PROGRAM Recipe13
VAR_INPUT
	ExecutingRecipe1: BOOL;
END_VAR
VAR_OUTPUT
	SuccesfullyEnded: BOOL := FALSE;
END_VAR
VAR
	State: INT := 0;
	WoodInitialLiftingPosition: INT := 50;
	InitialExtensionPosition: INT := 388;
	MaxGripPosition: INT := 160;
	RotationDropOffPosition: INT := 300;
	PlasticsInitialLiftingPosition: INT := 250;
	PlasticsDropOffExtensionPosition: INT := 300;
	MetalInitialLiftingPosition: INT := 400;
	MetalDropOffExtensionPosition: INT := 500;
END_VAR

// Recipe is sequence of moves to execute the task.

IF ExecutingRecipe1 THEN	// we start executing recipe1 (again)
	SuccesfullyEnded := FALSE;
END_IF

IF NOT IO.Switch AND NOT SuccesfullyEnded THEN
	IO.LEDGreen := 1;
	// WOOD:
	IF State = 0 THEN
		IF Automatic.LiftingPositionAuto < WoodInitialLiftingPosition THEN
			IO.MotorLiftingDirection := 0;
			IF NOT Automatic.SafetyLON THEN
				Automatic.MotorL.CurrentlyMoving := TRUE;
				IO.MotorLifting := 1;
			END_IF
		ELSE
			State := 1;
			IO.MotorLifting := 0;
			Automatic.MotorL.CurrentlyMoving := FALSE;
		END_IF
	ELSIF State = 1 THEN
		IF Automatic.ExtensionPositionAuto < InitialExtensionPosition THEN
			IO.MotorExtensionDirection := 0;
			IF NOT Automatic.SafetyEON THEN
				Automatic.MotorE.CurrentlyMoving := TRUE;
				IO.MotorExtension := 1;
			END_IF
		ELSE
			State := 2;
			IO.MotorExtension := 0;
			Automatic.MotorE.CurrentlyMoving := FALSE;
		END_IF
	ELSIF State = 2 THEN
		IF Automatic.GripPositionAuto < MaxGripPosition THEN
			IO.MotorGripDirection := 0;
			IF NOT Automatic.SafetyGON THEN
				Automatic.MotorG.CurrentlyMoving := TRUE;
				IO.MotorGrip := 1;
			END_IF
		ELSE
			State := 3;
			IO.MotorGrip := 0;
			Automatic.MotorG.CurrentlyMoving := FALSE;
		END_IF
	ELSIF State = 3 THEN
		IF NOT IO.EndLiftingSensor THEN
			IO.MotorLiftingDirection := 1;
			IF NOT Automatic.SafetyLON THEN
				Automatic.MotorG.CurrentlyMoving := TRUE;
				IO.MotorLifting := 1;
			END_IF
		ELSE
			State := 4;
			IO.MotorLifting := 0;
			Automatic.MotorL.CurrentlyMoving := FALSE;
		END_IF
	ELSIF State = 4 THEN
		IF Automatic.RotationPositionAuto < RotationDropOffPosition THEN
			IO.MotorRotationDirection := 0;
			IF NOT Automatic.SafetyRON THEN
				Automatic.MotorR.CurrentlyMoving := TRUE;
				IO.MotorRotation := 1;
			END_IF
		ELSE
			State := 5;
			IO.MotorRotation := 0;
			Automatic.MotorR.CurrentlyMoving := FALSE;
		END_IF
	ELSIF State = 5 THEN
		IF NOT IO.EndExtensionSensor THEN	// it drops wood in the nearest bin
			IO.MotorExtensionDirection := 1;
			IF NOT Automatic.SafetyEON THEN
				Automatic.MotorE.CurrentlyMoving := TRUE;
				IO.MotorExtension := 1;
			END_IF
		ELSE
			State := 6;
			IO.MotorExtension := 0;
			Automatic.MotorE.CurrentlyMoving := FALSE;
		END_IF
	ELSIF State = 6 THEN
		IF NOT IO.EndGripSensor THEN
			IO.MotorGripDirection := 1;
			IF NOT Automatic.SafetyGON THEN
				Automatic.MotorG.CurrentlyMoving := TRUE;
				IO.MotorGrip := 1;
			END_IF
		ELSE
			State := 7;
			IO.MotorGrip := 0;
			Automatic.MotorG.CurrentlyMoving := FALSE;
		END_IF
	ELSIF State = 7 THEN
		IF NOT IO.EndRotationSensor THEN
			IO.MotorRotationDirection := 1;
			IF NOT Automatic.SafetyRON THEN
				Automatic.MotorR.CurrentlyMoving := TRUE;
				IO.MotorRotation := 1;
			END_IF
		ELSE
			State := 8;
			IO.MotorRotation := 0;
			Automatic.MotorR.CurrentlyMoving := FALSE;
		END_IF
	END_IF
	
	// PLASTICS:
	IF State = 8 THEN
		IF Automatic.LiftingPositionAuto < PlasticsInitialLiftingPosition THEN
			IO.MotorLiftingDirection := 0;
			IF NOT Automatic.SafetyLON THEN
				Automatic.MotorL.CurrentlyMoving := TRUE;
				IO.MotorLifting := 1;
			END_IF
		ELSE
			State := 9;
			IO.MotorLifting := 0;
			Automatic.MotorL.CurrentlyMoving := FALSE;
		END_IF
	ELSIF State = 9 THEN
		IF Automatic.ExtensionPositionAuto < InitialExtensionPosition THEN
			IO.MotorExtensionDirection := 0;
			IF NOT Automatic.SafetyEON THEN
				Automatic.MotorE.CurrentlyMoving := TRUE;
				IO.MotorExtension := 1;
			END_IF
		ELSE
			State := 10;
			IO.MotorExtension := 0;
			Automatic.MotorE.CurrentlyMoving := FALSE;
		END_IF
	ELSIF State = 10 THEN
		IF Automatic.GripPositionAuto < MaxGripPosition THEN
			IO.MotorGripDirection := 0;
			IF NOT Automatic.SafetyGON THEN
				Automatic.MotorG.CurrentlyMoving := TRUE;
				IO.MotorGrip := 1;
			END_IF
		ELSE
			State := 11;
			IO.MotorGrip := 0;
			Automatic.MotorG.CurrentlyMoving := FALSE;
		END_IF
	ELSIF State = 11 THEN
		IF NOT IO.EndLiftingSensor THEN
			IO.MotorLiftingDirection := 1;
			IF NOT Automatic.SafetyLON THEN
				Automatic.MotorL.CurrentlyMoving := TRUE;
				IO.MotorLifting := 1;
			END_IF
		ELSE
			State := 12;
			IO.MotorLifting := 0;
			Automatic.MotorL.CurrentlyMoving := FALSE;
		END_IF
	ELSIF State = 12 THEN
		IF Automatic.RotationPositionAuto < RotationDropOffPosition THEN
			IO.MotorRotationDirection := 0;
			IF NOT Automatic.SafetyRON THEN
				Automatic.MotorR.CurrentlyMoving := TRUE;
				IO.MotorRotation := 1;
			END_IF
		ELSE
			State := 13;
			IO.MotorRotation := 0;
			Automatic.MotorR.CurrentlyMoving := FALSE;
		END_IF
	ELSIF State = 13 THEN
		IF Automatic.ExtensionPositionAuto > PlasticsDropOffExtensionPosition THEN	// it drops plastics into second nearest bin
			IO.MotorExtensionDirection := 1;
			IF NOT Automatic.SafetyEON THEN
				Automatic.MotorE.CurrentlyMoving := TRUE;
				IO.MotorExtension := 1;
			END_IF
		ELSE
			State := 14;
			IO.MotorExtension := 0;
			Automatic.MotorE.CurrentlyMoving := FALSE;
		END_IF
	ELSIF State = 14 THEN
		IF NOT IO.EndGripSensor THEN
			IO.MotorGripDirection := 1;
			IF NOT Automatic.SafetyGON THEN
				Automatic.MotorG.CurrentlyMoving := TRUE;
				IO.MotorGrip := 1;
			END_IF
		ELSE
			State := 15;
			IO.MotorGrip := 0;
			Automatic.MotorG.CurrentlyMoving := FALSE;
		END_IF
	ELSIF State = 15 THEN
		IF NOT IO.EndRotationSensor THEN
			IO.MotorRotationDirection := 1;
			IF NOT Automatic.SafetyRON THEN
				Automatic.MotorR.CurrentlyMoving := TRUE;
				IO.MotorRotation := 1;
			END_IF
		ELSE
			State := 16;
			IO.MotorRotation := 0;
			Automatic.MotorR.CurrentlyMoving := FALSE;
		END_IF
	END_IF
	
	// METAL:
	IF State = 16 THEN
		IF Automatic.LiftingPositionAuto < MetalInitialLiftingPosition THEN
			IO.MotorLiftingDirection := 0;
			IF NOT Automatic.SafetyLON THEN
				Automatic.MotorL.CurrentlyMoving := TRUE;
				IO.MotorLifting := 1;
			END_IF
		ELSE
			State := 17;
			IO.MotorLifting := 0;
			Automatic.MotorL.CurrentlyMoving := FALSE;
		END_IF
	ELSIF State = 17 THEN
		IF Automatic.ExtensionPositionAuto < InitialExtensionPosition THEN
			IO.MotorExtensionDirection := 0;
			IF NOT Automatic.SafetyEON THEN
				Automatic.MotorE.CurrentlyMoving := TRUE;
				IO.MotorExtension := 1;
			END_IF
		ELSE
			State := 18;
			IO.MotorExtension := 0;
			Automatic.MotorE.CurrentlyMoving := FALSE;
		END_IF
	ELSIF State = 18 THEN
		IF Automatic.GripPositionAuto < MaxGripPosition THEN
			IO.MotorGripDirection := 0;
			IF NOT Automatic.SafetyGON THEN
				Automatic.MotorG.CurrentlyMoving := TRUE;
				IO.MotorGrip := 1;
			END_IF
		ELSE
			State := 19;
			IO.MotorGrip := 0;
			Automatic.MotorG.CurrentlyMoving := FALSE;
		END_IF
	ELSIF State = 19 THEN
		IF NOT IO.EndLiftingSensor THEN
			IO.MotorLiftingDirection := 1;
			IF NOT Automatic.SafetyLON THEN
				Automatic.MotorL.CurrentlyMoving := TRUE;
				IO.MotorLifting := 1;
			END_IF
		ELSE
			State := 20;
			IO.MotorLifting := 0;
			Automatic.MotorL.CurrentlyMoving := FALSE;
		END_IF
	ELSIF State = 20 THEN
		IF Automatic.RotationPositionAuto < RotationDropOffPosition THEN
			IO.MotorRotationDirection := 0;
			IF NOT Automatic.SafetyRON THEN
				Automatic.MotorR.CurrentlyMoving := TRUE;
				IO.MotorRotation := 1;
			END_IF
		ELSE
			State := 21;
			IO.MotorRotation := 0;
			Automatic.MotorR.CurrentlyMoving := FALSE;
		END_IF
	ELSIF State = 21 THEN
		IF Automatic.ExtensionPositionAuto > MetalDropOffExtensionPosition THEN	// it drops metal into farthest bin
			IO.MotorExtensionDirection := 1;
			IF NOT Automatic.SafetyEON THEN
				Automatic.MotorE.CurrentlyMoving := TRUE;
				IO.MotorExtension := 1;
			END_IF
		ELSE
			State := 22;
			IO.MotorExtension := 0;
			Automatic.MotorE.CurrentlyMoving := FALSE;
		END_IF
	ELSIF State = 22 THEN
		IF NOT IO.EndGripSensor THEN
			IO.MotorGripDirection := 1;
			IF NOT Automatic.SafetyGON THEN
				Automatic.MotorG.CurrentlyMoving := TRUE;
				IO.MotorGrip := 1;
			END_IF
		ELSE
			State := 23;
			IO.MotorGrip := 0;
			Automatic.MotorG.CurrentlyMoving := FALSE;
		END_IF
	ELSIF State = 23 THEN
		IF NOT IO.EndRotationSensor THEN
			IO.MotorRotationDirection := 1;
			IF NOT Automatic.SafetyRON THEN
				Automatic.MotorR.CurrentlyMoving := TRUE;
				IO.MotorRotation := 1;
			END_IF
		ELSE
			State := 24;
			IO.MotorRotation := 0;
			Automatic.MotorR.CurrentlyMoving := FALSE;
		END_IF
	ELSIF State = 24 THEN
		SuccesfullyEnded := TRUE;
		State := 0;
		RETURN;
	END_IF
END_IF
RETURN;

END_PROGRAM

(* stored: Version 1.1.0.1, ProductVersion 3.1.4024.13
   POU Recipe13: Id {3098573e-c5b9-45cc-a6c2-48fae2f326e0}, SpecialFunc None *)
